TYPE ST_CN_CentralMachineCoolingDefaultParameters :
STRUCT
	///return temperature because feed temperature cannot be controlled
	aSetPointLimitsTemperature : ARRAY[1..2] OF REAL := [15,23];
END_STRUCT
END_TYPE

(* stored: Version 1.1.0.1, ProductVersion 3.1.4024.10
   DUT ST_CN_CentralMachineCoolingDefaultParameters: Id {17c81d14-e483-4b0e-9f64-7c549251bf40} *)
